FUNCTION_BLOCK FB_RecipeBuilderArona EXTENDS FB_RecipeBase

METHOD Build : BOOL
VAR_INST
    // Zmienne zostaną dodane w trakcie cyklu TDD
END_VAR
// ==========================================================
//  PLACEHOLDER / WYDMUSZKA - KOD DO ROZWOJU W TDD
// ==========================================================

// 1. Zabezpieczenie: Ustawiamy liczby segmentów na -1.
// Ponieważ 0 jest legalną wartością (np. program tylko do frezowania), 
// używamy -1 jako jednoznacznej flagi "brak implementacji".
_SegmentsToGroove := 2;
_SegmentsToCutX   := 2;
_SegmentsToCutY   := 2;

// TODO: Tutaj w TDD zaimplementujesz wyliczanie współrzędnych

// 2. Blokada przed uruchomieniem.
// W teście jednostkowym Twoja pierwsza asercja powinna sprawdzać 
// właśnie to, czy Builder.Build() zwrócił TRUE.
Build := TRUE;
END_METHOD

END_FUNCTION_BLOCK

(* stored: Version 1.1.0.1, ProductVersion 3.1.4024.15
   POU FB_RecipeBuilderArona: Id {a7865aba-34a9-4367-9b70-65119865d0af}, SpecialFunc None
   Method Build: Id {888409fe-0b8e-46d6-8abb-5ebdab25e661} *)
